PROGRAM MAIN
VAR
	fbIO	: FB_IOManager;
END_VAR

fbIO();

END_PROGRAM

(* stored: Version 1.1.0.1, ProductVersion 3.1.4024.12
   POU MAIN: Id {7c8913f8-ca68-46b0-869e-8df420903166}, SpecialFunc None *)
